// TIA Portal V17 export
// export: Created 2025-08-28T07:40:12.8284914Z, ExportSetting WithDefaults, DisplayName Totally Integrated Automation Portal, DisplayVersion V17, DisplayName TIA Portal Openness, DisplayVersion V17, DisplayName TIA Portal Version Control Interface, DisplayVersion V17, DisplayName STEP 7 Professional, DisplayVersion V17, DisplayName STEP 7 Safety, DisplayVersion V17, DisplayName WinCC Advanced, DisplayVersion V17
FUNCTION "energy_meter_read" : Void   // FC7, SCL
{ S7_Optimized_Access := 'TRUE' }
VERSION : 0.1
// stored: AutoNumber true, IsIECCheckEnabled false, SetENOAutomatically false, UDAEnableTagReadback false
BEGIN
   //读电能表数据

   //读电压
   //A相
   %DB2. := %DB5.;
   %DB2. := %DB5.;
   "local_control".energy_meter[0] := "local_control".energy_meter[0] / 10.0;

   //读电压
   //B相
   %DB2. := %DB5.;
   %DB2. := %DB5.;
   "local_control".energy_meter[1] := "local_control".energy_meter[1] / 10.0;

   //读电压
   //C相
   %DB2. := %DB5.;
   %DB2. := %DB5.;
   "local_control".energy_meter[2] := "local_control".energy_meter[2] / 10.0;

   //读电流
   //A相
   %DB2. := %DB5.;
   %DB2. := %DB5.;
   "local_control".energy_meter[3] := "local_control".energy_meter[3] / 1000.0;

   //读电流
   //B相
   %DB2. := %DB5.;
   %DB2. := %DB5.;
   "local_control".energy_meter[4] := "local_control".energy_meter[4] / 1000.0;

   //读电流
   //C相
   %DB2. := %DB5.;
   %DB2. := %DB5.;
   "local_control".energy_meter[5] := "local_control".energy_meter[5] / 1000.0;

   //读电能
   //正向有功总电能
   %DB2. := %DB5.;
   %DB2. := %DB5.;
   "local_control".energy_meter[6] := "local_control".energy_meter[6] / 10.0;
END_FUNCTION
